% RSLogix 500 project Hopper_DIGI_P2_showcase2.RSS, saved by version 8.30.00.16 %
PROJECT "UNTITLED"    % processor: Bul.1763 MicroLogix 1100 Series A %

PROGRAM FILES
  LAD 2 "MAIN"  3 rungs
  LAD 3 "I/O"  5 rungs
  LAD 4 "CONTROLS"  6 rungs

DATA FILES
  O0 OUTPUT  5 elements
  I1 INPUT  7 elements
  S2 STATUS  66 elements
  B3 BINARY  2 elements
  T4 TIMER  1 elements
  C5 COUNTER  1 elements
  R6 CONTROL  1 elements
  N7 INTEGER  1 elements
  F8 FLOAT  1 elements

LADDER 2 "MAIN"
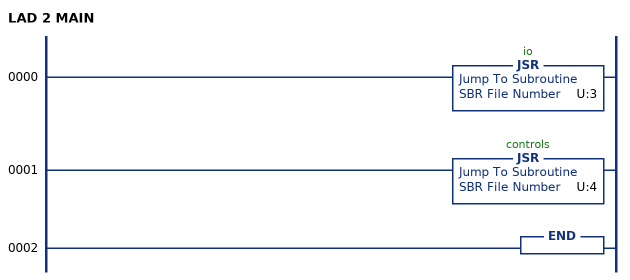
% Rung: 0 %
SOR JSR U:3 EOR
%   U:3  "io" %
% Rung: 1 %
SOR JSR U:4 EOR
%   U:4  "controls" %
% Rung: 2 %
SOR END EOR

LADDER 3 "I/O"
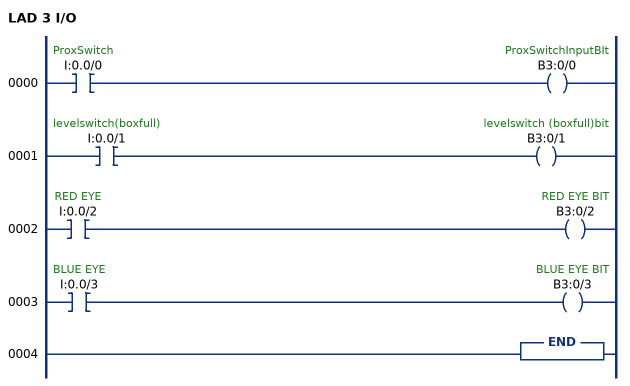
% Rung: 0 %
SOR XIC I:0.0/0 OTE B3:0/0 EOR
%   I:0.0/0  "ProxSwitch" %
%   B3:0/0  "ProxSwitchInputBIt" %
% Rung: 1 %
SOR XIC I:0.0/1 OTE B3:0/1 EOR
%   I:0.0/1  "levelswitch(boxfull)" %
%   B3:0/1  "levelswitch (boxfull)bit" %
% Rung: 2 %
SOR XIC I:0.0/2 OTE B3:0/2 EOR
%   I:0.0/2  "RED EYE" %
%   B3:0/2  "RED EYE BIT" %
% Rung: 3 %
SOR XIC I:0.0/3 OTE B3:0/3 EOR
%   I:0.0/3  "BLUE EYE" %
%   B3:0/3  "BLUE EYE BIT" %
% Rung: 4 %
SOR END EOR

LADDER 4 "CONTROLS"
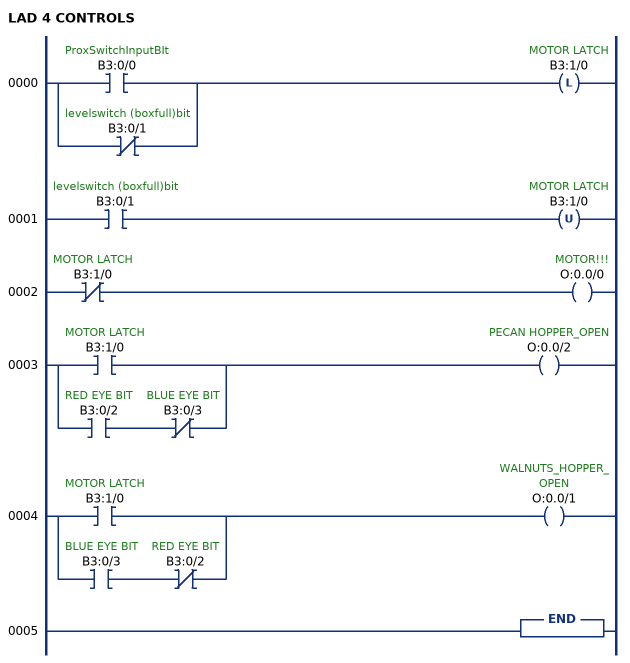
% Rung: 0 %  % edit flag set %
SOR BST XIC B3:0/0 NXB XIO B3:0/1 BND OTL B3:1/0 EOR
%   B3:0/0  "ProxSwitchInputBIt" %
%   B3:0/1  "levelswitch (boxfull)bit" %
%   B3:1/0  "MOTOR LATCH" %
% Rung: 1 %
SOR XIC B3:0/1 OTU B3:1/0 EOR
%   B3:0/1  "levelswitch (boxfull)bit" %
%   B3:1/0  "MOTOR LATCH" %
% Rung: 2 %
SOR XIO B3:1/0 OTE O:0.0/0 EOR
%   B3:1/0  "MOTOR LATCH" %
%   O:0.0/0  "MOTOR!!!" %
% Rung: 3 %
SOR BST XIC B3:1/0 NXB XIC B3:0/2 XIO B3:0/3 BND OTE O:0.0/2 EOR
%   B3:1/0  "MOTOR LATCH" %
%   B3:0/2  "RED EYE BIT" %
%   B3:0/3  "BLUE EYE BIT" %
%   O:0.0/2  "PECAN HOPPER_OPEN" %
% Rung: 4 %
SOR BST XIC B3:1/0 NXB XIC B3:0/3 XIO B3:0/2 BND OTE O:0.0/1 EOR
%   B3:1/0  "MOTOR LATCH" %
%   B3:0/3  "BLUE EYE BIT" %
%   B3:0/2  "RED EYE BIT" %
%   O:0.0/1  "WALNUTS_HOPPER_OPEN" %
% Rung: 5 %
SOR END EOR

REVISION NOTES
  0: test2
